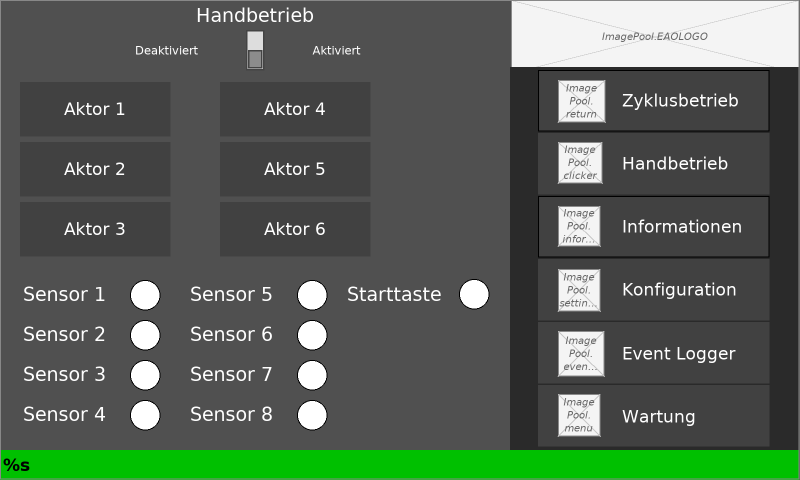
VISUALIZATION Handbetrieb  // 800x480
    Image (511,0 288x73), image: ImagePool.EAOLOGO
    Rectangle (510,67 289x412)
    Textfield (155,1 200x29), "Handbetrieb"
    Textfield (130,25 73x51), "Deaktiviert"
    Textfield (300,25 73x51), "Aktiviert"
    Rectangle (0,450 799x30), "%s", text variable: MAIN.HMI.sStatus, colour variable: MAIN.HMI.nColorInfoBalken
        p3450524324: MAIN.HMI.nColorInfoBalken
    DipSwitch (210,30 90x40), variable: MAIN.bE_Handbetrieb, behaviour: TOGGLE, style: Switch-DipSwitch-Gray
    Textfield (20,82 150x54), "Aktor 1", colour toggle: MAIN.fbSt1.fbAktor[1].bA_arbeitsPos
        OnMouseClick: execute { MAIN.fbSt1.fbAktor[1].bBtnHandausloesung := TRUE; }
    Textfield (20,142 150x54), "Aktor 2", colour toggle: MAIN.fbSt1.fbAktor[2].bA_arbeitsPos
        OnMouseClick: execute { MAIN.fbSt1.fbAktor[2].bBtnHandausloesung := TRUE; }
    Rectangle (538,70 231x61)
        OnMouseClick: change screen: Zyklusbetrieb
    Textfield (619,70 153x61), "Zyklusbetrieb"
        OnMouseClick: change screen: Zyklusbetrieb
    Rectangle (538,133 231x61)
        OnMouseClick: change screen: Handbetrieb
    Textfield (619,133 153x61), "Handbetrieb"
        OnMouseClick: change screen: Handbetrieb
    Image (558,142 44x41), image: ImagePool.clicker
        OnMouseClick: change screen: Handbetrieb
    Image (558,80 47x42), image: ImagePool.return
        OnMouseClick: change screen: Zyklusbetrieb
    Rectangle (538,196 231x61)
        OnMouseClick: change screen: Diagnose
    Textfield (619,196 153x61), "Informationen"
        OnMouseClick: change screen: Diagnose
    Image (558,206 42x40), image: ImagePool.information
        OnMouseClick: change screen: Diagnose
    Rectangle (538,322 231x61)
        OnMouseClick: change screen: EventLogger
    Textfield (619,323 153x61), "Event Logger"
        OnMouseClick: change screen: EventLogger
    Image (558,331 46x45), image: ImagePool.eventLogger
        OnMouseClick: change screen: EventLogger
    Rectangle (538,259 231x61)
        OnMouseClick: change screen: Konfig1
    Textfield (619,259 153x61), "Konfiguration"
        OnMouseClick: change screen: Konfig1
    Image (558,269 42x42), image: ImagePool.settings
        OnMouseDown: change screen: Konfig1
    Rectangle (538,385 231x61)
        OnMouseClick: change screen: Wartung
    Textfield (619,386 153x61), "Wartung"
        OnMouseClick: change screen: Wartung
    Image (558,394 42x42), image: ImagePool.menu
        OnMouseDown: change screen: Wartung
    Textfield (20,202 150x54), "Aktor 3", colour toggle: MAIN.fbSt1.fbAktor[3].bA_arbeitsPos
        OnMouseClick: execute { MAIN.fbSt1.fbAktor[3].bBtnHandausloesung := TRUE; }
    Textfield (220,82 150x54), "Aktor 4", colour toggle: MAIN.fbSt1.fbAktor[4].bA_arbeitsPos
        OnMouseClick: execute { MAIN.fbSt1.fbAktor[4].bBtnHandausloesung := TRUE; }
    Textfield (220,142 150x54), "Aktor 5", colour toggle: MAIN.fbSt1.fbAktor[5].bA_arbeitsPos
        OnMouseClick: execute { MAIN.fbSt1.fbAktor[5].bBtnHandausloesung := TRUE; }
    Textfield (220,202 150x54), "Aktor 6", colour toggle: MAIN.fbSt1.fbAktor[6].bA_arbeitsPos
        OnMouseClick: execute { MAIN.fbSt1.fbAktor[6].bBtnHandausloesung := TRUE; }
    Textfield (20,280 123x29), "Sensor 1"
    Textfield (187,280 123x29), "Sensor 5"
    Textfield (20,320 123x29), "Sensor 2"
    Textfield (187,320 123x29), "Sensor 6"
    Textfield (20,360 123x29), "Sensor 3"
    Textfield (187,360 123x29), "Sensor 7"
    Textfield (187,400 123x29), "Sensor 8"
    Textfield (20,400 123x29), "Sensor 4"
    Ellipse (130,280 30x30), colour toggle: MAIN.fbSt1.bE_Sensor[1]
    Ellipse (130,320 30x30), colour toggle: MAIN.fbSt1.bE_Sensor[2]
    Ellipse (130,360 30x30), colour toggle: MAIN.fbSt1.bE_Sensor[3]
    Ellipse (130,400 30x30), colour toggle: MAIN.fbSt1.bE_Sensor[4]
    Ellipse (297,320 30x30), colour toggle: MAIN.fbSt1.bE_Sensor[6]
    Ellipse (297,280 30x30), colour toggle: MAIN.fbSt1.bE_Sensor[5]
    Ellipse (297,360 30x30), colour toggle: MAIN.fbSt1.bE_Sensor[7]
    Ellipse (297,400 30x30), colour toggle: MAIN.fbSt1.bE_Sensor[8]
    Textfield (344,280 123x29), "Starttaste"
    Ellipse (459,279 30x30), colour toggle: MAIN.bE_Fussschalter
END_VISUALIZATION

(* stored: Version 1.1.0.1, ProductVersion 3.1.4024.12
   Visu Handbetrieb: Id {42aa99ba-a1b4-4978-b2eb-52b07b27a7b2} *)
